{attribute 'GeneratedUsingTerminal: EK1100-0000-0018'}
{attribute addProperty BoxType "EK1100-0000-0018"}
{attribute addProperty Id "Beckhoff_EL1xxxEK1122Beckhoff_EL1xxxEK1122_4D1603AD2A_0001_EL1002_0000_0000EL1002_02444DCB6A_0002_EL1002_0000_0016EL1002_02444DCB6A_0003_EL1002_0000_0017EL1002_02444DCB6A_0004_EL1002_0000_0018EL1002_02444DCB6A_0005_EL1004_0000_0000EL1004_D135F8DB8A_0006_EL1004_0000_0016EL1004_D135F8DB8A_0007_EL1004_0000_0017EL1004_D135F8DB8A_0008_EL1004_0000_0018EL1004_D135F8DB8A_0009_EL1004_0000_0019EL1004_D135F8DB8A_0010_EL1004_0010_0000EL1004_D135F8DB8A_0011_EL1004_0010_0016EL1004_D135F8DB8A_0012_EL1004_0010_0017EL1004_D135F8DB8A_0013_EL1004_0010_0018EL1004_D135F8DB8A_0014_EL1004_0020_0016EL1004_D135F8DB8A_0015_EL1008_0000_0016EL1008_78E8D3DD12A_0016_EL1008_0000_0017EL1008_78E8D3DD12A_0017_EL1008_0000_0018EL1008_78E8D3DD12A_0018_EL1012_0000_0000EL1012_02444DCB6A_0019_EL1012_0000_0016EL1012_02444DCB6A_0020_EL1012_0000_0017EL1012_02444DCB6A_0021_EL1012_0000_0018EL1012_02444DCB6A_0022_EL1014_0000_0000EL1014_D135F8DB8A_0023_EL1014_0000_0016EL1014_D135F8DB8A_0024_EL1014_0000_0017EL1014_D135F8DB8A_0025_EL1014_0000_0018EL1014_D135F8DB8A_0026_EL1014_0000_0019EL1014_D135F8DB8A_0027_EL1014_0010_0000EL1014_D135F8DB8A_0028_EL1014_0010_0016EL1014_D135F8DB8A_0029_EL1014_0010_0017EL1014_D135F8DB8A_0030_EL1014_0010_0018EL1014_D135F8DB8A_0031_EL1014_0010_0019EL1014_D135F8DB8A_0032_EL1018_0000_0016EL1018_78E8D3DD12A_0033_EL1018_0000_0017EL1018_78E8D3DD12A_0034_EL1018_0000_0018EL1018_78E8D3DD12A_0035_EL1024_0000_0016EL1024_D135F8DB8A_0036_EL1024_0000_0017EL1024_D135F8DB8A_0037_EL1024_0000_0018EL1024_D135F8DB8A_0038_EL1034_0000_0016EL1034_D135F8DB8A_0039_EL1034_0000_0017EL1034_D135F8DB8A_0040_EL1034_0000_0018EL1034_D135F8DB8A_0041_EL1052_0000_0016EL1052_6CC2DB6A8A_0042_EL1054_0000_0016EL1054_37C87A1C12A_0043_EL1084_0000_0016EL1084_D135F8DB8A_0044_EL1084_0000_0017EL1084_D135F8DB8A_0045_EL1084_0000_0018EL1084_D135F8DB8A_0046_EL1088_0000_0016EL1088_78E8D3DD12A_0047_EL1088_0000_0017EL1088_78E8D3DD12A_0048_EL1088_0000_0018EL1088_78E8D3DD12A_0049_EL1094_0000_0016EL1094_D135F8DB8A_0050_EL1094_0000_0017EL1094_D135F8DB8A_0051_EL1094_0000_0018EL1094_D135F8DB8A_0052_EL1098_0000_0016EL1098_78E8D3DD12A_0053_EL1098_0000_0017EL1098_78E8D3DD12A_0054_EL1098_0000_0018EL1098_78E8D3DD12A_0055_EL1104_0000_0016EL1104_D135F8DB8A_0056_EL1104_0000_0017EL1104_D135F8DB8A_0057_EL1104_0000_0018EL1104_D135F8DB8A_0058_EL1114_0000_0016EL1114_D135F8DB8A_0059_EL1114_0000_0017EL1114_D135F8DB8A_0060_EL1114_0000_0018EL1114_D135F8DB8A_0061_EL1124_0000_0016EL1124_D135F8DB8A_0062_EL1124_0000_0017EL1124_D135F8DB8A_0063_EL1124_0000_0018EL1124_D135F8DB8A_0064_EL1134_0000_0016EL1134_D135F8DB8A_0065_EL1134_0000_0017EL1134_D135F8DB8A_0066_EL1134_0000_0018EL1134_D135F8DB8A_0067_EL1144_0000_0016EL1144_D135F8DB8A_0068_EL1144_0000_0017EL1144_D135F8DB8A_0069_EL1144_0000_0018EL1144_D135F8DB8A_0070_EL1202_0000_0016EL1202_02444DCB6A_0071_EL1202_0000_0017EL1202_02444DCB6A_0072_EL1202_0000_0018EL1202_02444DCB6A_0073_EL1202_0000_0019EL1202_02444DCB6A_0074_EL1202_0100_0016EL1202_647E460722A_0075_EL1202_0100_0017EL1202_647E460722A_0076_EL1202_0100_0018EL1202_647E460722A_0077_EL1202_0100_0019EL1202_647E460722A_0078_EL1252_0000_0017EL1252_0C2D47B448A_0079_EL1252_0000_0018EL1252_934A18FC48A_0080_EL1252_0000_0019EL1252_934A18FC48A_0081_EL1252_0000_0020EL1252_934A18FC48A_0082_EL1252_0000_0021EL1252_934A18FC48A_0083_EL1252_0000_0022EL1252_934A18FC48A_0084_EL1252_0010_0019EL1252_934A18FC48A_0085_EL1252_0010_0020EL1252_934A18FC48A_0086_EL1252_0010_0021EL1252_934A18FC48A_0087_EL1252_0050_0016EL1252_934A18FC48A_0088_EL1252_0050_0017EL1252_934A18FC48A_0089_EL1252_0050_0018EL1252_934A18FC48A_0090_EL1254_0000_0000EL1254_D5E6FA5F84A_0091_EL1262_0000_0002EL1262_0FA571DE40A_0092_EL1262_0000_0003EL1262_0FA571DE40A_0093_EL1262_0050_0002EL1262_0FA571DE40A_0094_EL1262_0050_0003EL1262_0FA571DE40A_0095_EL1258_0000_0016EL1258_FA676B82476A_0096_EL1258_0000_0017EL1258_FA676B82476A_0097_EL1258_0010_0017EL1258_E0C61872116A_0098_EL1259_0000_0016EL1259_D83D5EFD964A_0099_EL1259_0000_0017EL1259_22458C8C972A_0100_EL1259_0000_0018EL1259_22458C8C972A_0101_EL1382_0000_0016EL1382_6CC2DB6A8A_0102_EL1382_0000_0017EL1382_6CC2DB6A8A_0103_EL1382_0000_0018EL1382_6CC2DB6A8A_0104_EL1702_0000_0016EL1702_02444DCB6A_0105_EL1702_0000_0017EL1702_02444DCB6A_0106_EL1702_0020_0016EL1702_02444DCB6A_0107_EL1712_0000_0016EL1712_02444DCB6A_0108_EL1712_0020_0016EL1712_02444DCB6A_0109_EL1722_0000_0016EL1722_02444DCB6A_0110_EL1722_0000_0017EL1722_02444DCB6A_0111_EL1804_0000_0016EL1804_D135F8DB8A_0112_EL1804_0000_0017EL1804_D135F8DB8A_0113_EL1804_0000_0018EL1804_D135F8DB8A_0114_EL1808_0000_0016EL1808_78E8D3DD12A_0115_EL1808_0000_0017EL1808_78E8D3DD12A_0116_EL1808_0000_0018EL1808_78E8D3DD12A_0117_EL1809_0000_0016EL1809_32157CFD20A_0118_EL1809_0000_0017EL1809_32157CFD20A_0119_EL1809_0000_0018EL1809_32157CFD20A_0120_EL1814_0000_0016EL1814_D135F8DB8A_0121_EL1814_0000_0017EL1814_D135F8DB8A_0122_EL1814_0000_0018EL1814_D135F8DB8A_0123_EL1819_0000_0016EL1819_32157CFD20A_0124_EL1819_0000_0017EL1819_32157CFD20A_0125_EL1819_0000_0018EL1819_32157CFD20A_0126_EL1852_0000_0016EL1852_7699BCF620A_0127_EL1859_0000_0016EL1859_7699BCF620A_0128_EL1859_0000_0017EL1859_7699BCF620A_0129_EL1859_0000_0018EL1859_7699BCF620A_0130_EL1862_0000_0016EL1862_32157CFD20A_0131_EL1862_0000_0017EL1862_32157CFD20A_0132_EL1862_0000_0018EL1862_32157CFD20A_0133_EL1862_0000_0019EL1862_32157CFD20A_0134_EL1862_0010_0016EL1862_32157CFD20A_0135_EL1862_0010_0017EL1862_32157CFD20A_0136_EL1862_0010_0018EL1862_32157CFD20A_0137_EL1862_0010_0019EL1862_32157CFD20A_0138_EL1872_0000_0016EL1872_32157CFD20A_0139_EL1872_0000_0017EL1872_32157CFD20A_0140_EL1872_0000_0018EL1872_32157CFD20A_0141_EL1872_0010_0016EL1872_32157CFD20A_0142_EL1889_0000_0016EL1889_32157CFD20A_0143_EL1889_0000_0017EL1889_32157CFD20A_0144_EL1889_0000_0018EL1889_32157CFD20A_0145_EL1889_0000_0019EL1889_32157CFD20A_0146_EL1899_0000_0016EL1899_32157CFD20"}
{attribute addProperty CRC "3845396967"}
{attribute addProperty Size "6188"}
TYPE Beckhoff_EL1xxx_E53419E7 EXTENDS EK1100_1FC0878B :
STRUCT
	{attribute addProperty Name "Beckhoff_EL1xxxEK1122"}
	{attribute addProperty PreviousPort "Beckhoff EL1xxx : B"}
	Beckhoff_EL1xxxEK1122 : Beckhoff_EL1xxxEK1122_4D1603AD;
	{attribute addProperty Name "A_0001_EL1002_0000_0000"}
	{attribute addProperty PreviousPort "Beckhoff EL1xxxEK1122 : C"}
	A_0001_EL1002_0000_0000 : EL1002_02444DCB;
	{attribute addProperty Name "A_0002_EL1002_0000_0016"}
	{attribute addProperty PreviousPort "A_0001(EL1002-0000-0000) : B"}
	A_0002_EL1002_0000_0016 : EL1002_02444DCB;
	{attribute addProperty Name "A_0003_EL1002_0000_0017"}
	{attribute addProperty PreviousPort "A_0002(EL1002-0000-0016) : B"}
	A_0003_EL1002_0000_0017 : EL1002_02444DCB;
	{attribute addProperty Name "A_0004_EL1002_0000_0018"}
	{attribute addProperty PreviousPort "A_0003(EL1002-0000-0017) : B"}
	A_0004_EL1002_0000_0018 : EL1002_02444DCB;
	{attribute addProperty Name "A_0005_EL1004_0000_0000"}
	{attribute addProperty PreviousPort "A_0004(EL1002-0000-0018) : B"}
	A_0005_EL1004_0000_0000 : EL1004_D135F8DB;
	{attribute addProperty Name "A_0006_EL1004_0000_0016"}
	{attribute addProperty PreviousPort "A_0005(EL1004-0000-0000) : B"}
	A_0006_EL1004_0000_0016 : EL1004_D135F8DB;
	{attribute addProperty Name "A_0007_EL1004_0000_0017"}
	{attribute addProperty PreviousPort "A_0006(EL1004-0000-0016) : B"}
	A_0007_EL1004_0000_0017 : EL1004_D135F8DB;
	{attribute addProperty Name "A_0008_EL1004_0000_0018"}
	{attribute addProperty PreviousPort "A_0007(EL1004-0000-0017) : B"}
	A_0008_EL1004_0000_0018 : EL1004_D135F8DB;
	{attribute addProperty Name "A_0009_EL1004_0000_0019"}
	{attribute addProperty PreviousPort "A_0008(EL1004-0000-0018) : B"}
	A_0009_EL1004_0000_0019 : EL1004_D135F8DB;
	{attribute addProperty Name "A_0010_EL1004_0010_0000"}
	{attribute addProperty PreviousPort "A_0009(EL1004-0000-0019) : B"}
	A_0010_EL1004_0010_0000 : EL1004_D135F8DB;
	{attribute addProperty Name "A_0011_EL1004_0010_0016"}
	{attribute addProperty PreviousPort "A_0010(EL1004-0010-0000) : B"}
	A_0011_EL1004_0010_0016 : EL1004_D135F8DB;
	{attribute addProperty Name "A_0012_EL1004_0010_0017"}
	{attribute addProperty PreviousPort "A_0011(EL1004-0010-0016) : B"}
	A_0012_EL1004_0010_0017 : EL1004_D135F8DB;
	{attribute addProperty Name "A_0013_EL1004_0010_0018"}
	{attribute addProperty PreviousPort "A_0012(EL1004-0010-0017) : B"}
	A_0013_EL1004_0010_0018 : EL1004_D135F8DB;
	{attribute addProperty Name "A_0014_EL1004_0020_0016"}
	{attribute addProperty PreviousPort "A_0013(EL1004-0010-0018) : B"}
	A_0014_EL1004_0020_0016 : EL1004_D135F8DB;
	{attribute addProperty Name "A_0015_EL1008_0000_0016"}
	{attribute addProperty PreviousPort "A_0014(EL1004-0020-0016) : B"}
	A_0015_EL1008_0000_0016 : EL1008_78E8D3DD;
	{attribute addProperty Name "A_0016_EL1008_0000_0017"}
	{attribute addProperty PreviousPort "A_0015(EL1008-0000-0016) : B"}
	A_0016_EL1008_0000_0017 : EL1008_78E8D3DD;
	{attribute addProperty Name "A_0017_EL1008_0000_0018"}
	{attribute addProperty PreviousPort "A_0016(EL1008-0000-0017) : B"}
	A_0017_EL1008_0000_0018 : EL1008_78E8D3DD;
	{attribute addProperty Name "A_0018_EL1012_0000_0000"}
	{attribute addProperty PreviousPort "A_0017(EL1008-0000-0018) : B"}
	A_0018_EL1012_0000_0000 : EL1012_02444DCB;
	{attribute addProperty Name "A_0019_EL1012_0000_0016"}
	{attribute addProperty PreviousPort "A_0018(EL1012-0000-0000) : B"}
	A_0019_EL1012_0000_0016 : EL1012_02444DCB;
	{attribute addProperty Name "A_0020_EL1012_0000_0017"}
	{attribute addProperty PreviousPort "A_0019(EL1012-0000-0016) : B"}
	A_0020_EL1012_0000_0017 : EL1012_02444DCB;
	{attribute addProperty Name "A_0021_EL1012_0000_0018"}
	{attribute addProperty PreviousPort "A_0020(EL1012-0000-0017) : B"}
	A_0021_EL1012_0000_0018 : EL1012_02444DCB;
	{attribute addProperty Name "A_0022_EL1014_0000_0000"}
	{attribute addProperty PreviousPort "A_0021(EL1012-0000-0018) : B"}
	A_0022_EL1014_0000_0000 : EL1014_D135F8DB;
	{attribute addProperty Name "A_0023_EL1014_0000_0016"}
	{attribute addProperty PreviousPort "A_0022(EL1014-0000-0000) : B"}
	A_0023_EL1014_0000_0016 : EL1014_D135F8DB;
	{attribute addProperty Name "A_0024_EL1014_0000_0017"}
	{attribute addProperty PreviousPort "A_0023(EL1014-0000-0016) : B"}
	A_0024_EL1014_0000_0017 : EL1014_D135F8DB;
	{attribute addProperty Name "A_0025_EL1014_0000_0018"}
	{attribute addProperty PreviousPort "A_0024(EL1014-0000-0017) : B"}
	A_0025_EL1014_0000_0018 : EL1014_D135F8DB;
	{attribute addProperty Name "A_0026_EL1014_0000_0019"}
	{attribute addProperty PreviousPort "A_0025(EL1014-0000-0018) : B"}
	A_0026_EL1014_0000_0019 : EL1014_D135F8DB;
	{attribute addProperty Name "A_0027_EL1014_0010_0000"}
	{attribute addProperty PreviousPort "A_0026(EL1014-0000-0019) : B"}
	A_0027_EL1014_0010_0000 : EL1014_D135F8DB;
	{attribute addProperty Name "A_0028_EL1014_0010_0016"}
	{attribute addProperty PreviousPort "A_0027(EL1014-0010-0000) : B"}
	A_0028_EL1014_0010_0016 : EL1014_D135F8DB;
	{attribute addProperty Name "A_0029_EL1014_0010_0017"}
	{attribute addProperty PreviousPort "A_0028(EL1014-0010-0016) : B"}
	A_0029_EL1014_0010_0017 : EL1014_D135F8DB;
	{attribute addProperty Name "A_0030_EL1014_0010_0018"}
	{attribute addProperty PreviousPort "A_0029(EL1014-0010-0017) : B"}
	A_0030_EL1014_0010_0018 : EL1014_D135F8DB;
	{attribute addProperty Name "A_0031_EL1014_0010_0019"}
	{attribute addProperty PreviousPort "A_0030(EL1014-0010-0018) : B"}
	A_0031_EL1014_0010_0019 : EL1014_D135F8DB;
	{attribute addProperty Name "A_0032_EL1018_0000_0016"}
	{attribute addProperty PreviousPort "A_0031(EL1014-0010-0019) : B"}
	A_0032_EL1018_0000_0016 : EL1018_78E8D3DD;
	{attribute addProperty Name "A_0033_EL1018_0000_0017"}
	{attribute addProperty PreviousPort "A_0032(EL1018-0000-0016) : B"}
	A_0033_EL1018_0000_0017 : EL1018_78E8D3DD;
	{attribute addProperty Name "A_0034_EL1018_0000_0018"}
	{attribute addProperty PreviousPort "A_0033(EL1018-0000-0017) : B"}
	A_0034_EL1018_0000_0018 : EL1018_78E8D3DD;
	{attribute addProperty Name "A_0035_EL1024_0000_0016"}
	{attribute addProperty PreviousPort "A_0034(EL1018-0000-0018) : B"}
	A_0035_EL1024_0000_0016 : EL1024_D135F8DB;
	{attribute addProperty Name "A_0036_EL1024_0000_0017"}
	{attribute addProperty PreviousPort "A_0035(EL1024-0000-0016) : B"}
	A_0036_EL1024_0000_0017 : EL1024_D135F8DB;
	{attribute addProperty Name "A_0037_EL1024_0000_0018"}
	{attribute addProperty PreviousPort "A_0036(EL1024-0000-0017) : B"}
	A_0037_EL1024_0000_0018 : EL1024_D135F8DB;
	{attribute addProperty Name "A_0038_EL1034_0000_0016"}
	{attribute addProperty PreviousPort "A_0037(EL1024-0000-0018) : B"}
	A_0038_EL1034_0000_0016 : EL1034_D135F8DB;
	{attribute addProperty Name "A_0039_EL1034_0000_0017"}
	{attribute addProperty PreviousPort "A_0038(EL1034-0000-0016) : B"}
	A_0039_EL1034_0000_0017 : EL1034_D135F8DB;
	{attribute addProperty Name "A_0040_EL1034_0000_0018"}
	{attribute addProperty PreviousPort "A_0039(EL1034-0000-0017) : B"}
	A_0040_EL1034_0000_0018 : EL1034_D135F8DB;
	{attribute addProperty Name "A_0041_EL1052_0000_0016"}
	{attribute addProperty PreviousPort "A_0040(EL1034-0000-0018) : B"}
	A_0041_EL1052_0000_0016 : EL1052_6CC2DB6A;
	{attribute addProperty Name "A_0042_EL1054_0000_0016"}
	{attribute addProperty PreviousPort "A_0041(EL1052-0000-0016) : B"}
	A_0042_EL1054_0000_0016 : EL1054_37C87A1C;
	{attribute addProperty Name "A_0043_EL1084_0000_0016"}
	{attribute addProperty PreviousPort "A_0042(EL1054-0000-0016) : B"}
	A_0043_EL1084_0000_0016 : EL1084_D135F8DB;
	{attribute addProperty Name "A_0044_EL1084_0000_0017"}
	{attribute addProperty PreviousPort "A_0043(EL1084-0000-0016) : B"}
	A_0044_EL1084_0000_0017 : EL1084_D135F8DB;
	{attribute addProperty Name "A_0045_EL1084_0000_0018"}
	{attribute addProperty PreviousPort "A_0044(EL1084-0000-0017) : B"}
	A_0045_EL1084_0000_0018 : EL1084_D135F8DB;
	{attribute addProperty Name "A_0046_EL1088_0000_0016"}
	{attribute addProperty PreviousPort "A_0045(EL1084-0000-0018) : B"}
	A_0046_EL1088_0000_0016 : EL1088_78E8D3DD;
	{attribute addProperty Name "A_0047_EL1088_0000_0017"}
	{attribute addProperty PreviousPort "A_0046(EL1088-0000-0016) : B"}
	A_0047_EL1088_0000_0017 : EL1088_78E8D3DD;
	{attribute addProperty Name "A_0048_EL1088_0000_0018"}
	{attribute addProperty PreviousPort "A_0047(EL1088-0000-0017) : B"}
	A_0048_EL1088_0000_0018 : EL1088_78E8D3DD;
	{attribute addProperty Name "A_0049_EL1094_0000_0016"}
	{attribute addProperty PreviousPort "A_0048(EL1088-0000-0018) : B"}
	A_0049_EL1094_0000_0016 : EL1094_D135F8DB;
	{attribute addProperty Name "A_0050_EL1094_0000_0017"}
	{attribute addProperty PreviousPort "A_0049(EL1094-0000-0016) : B"}
	A_0050_EL1094_0000_0017 : EL1094_D135F8DB;
	{attribute addProperty Name "A_0051_EL1094_0000_0018"}
	{attribute addProperty PreviousPort "A_0050(EL1094-0000-0017) : B"}
	A_0051_EL1094_0000_0018 : EL1094_D135F8DB;
	{attribute addProperty Name "A_0052_EL1098_0000_0016"}
	{attribute addProperty PreviousPort "A_0051(EL1094-0000-0018) : B"}
	A_0052_EL1098_0000_0016 : EL1098_78E8D3DD;
	{attribute addProperty Name "A_0053_EL1098_0000_0017"}
	{attribute addProperty PreviousPort "A_0052(EL1098-0000-0016) : B"}
	A_0053_EL1098_0000_0017 : EL1098_78E8D3DD;
	{attribute addProperty Name "A_0054_EL1098_0000_0018"}
	{attribute addProperty PreviousPort "A_0053(EL1098-0000-0017) : B"}
	A_0054_EL1098_0000_0018 : EL1098_78E8D3DD;
	{attribute addProperty Name "A_0055_EL1104_0000_0016"}
	{attribute addProperty PreviousPort "A_0054(EL1098-0000-0018) : B"}
	A_0055_EL1104_0000_0016 : EL1104_D135F8DB;
	{attribute addProperty Name "A_0056_EL1104_0000_0017"}
	{attribute addProperty PreviousPort "A_0055(EL1104-0000-0016) : B"}
	A_0056_EL1104_0000_0017 : EL1104_D135F8DB;
	{attribute addProperty Name "A_0057_EL1104_0000_0018"}
	{attribute addProperty PreviousPort "A_0056(EL1104-0000-0017) : B"}
	A_0057_EL1104_0000_0018 : EL1104_D135F8DB;
	{attribute addProperty Name "A_0058_EL1114_0000_0016"}
	{attribute addProperty PreviousPort "A_0057(EL1104-0000-0018) : B"}
	A_0058_EL1114_0000_0016 : EL1114_D135F8DB;
	{attribute addProperty Name "A_0059_EL1114_0000_0017"}
	{attribute addProperty PreviousPort "A_0058(EL1114-0000-0016) : B"}
	A_0059_EL1114_0000_0017 : EL1114_D135F8DB;
	{attribute addProperty Name "A_0060_EL1114_0000_0018"}
	{attribute addProperty PreviousPort "A_0059(EL1114-0000-0017) : B"}
	A_0060_EL1114_0000_0018 : EL1114_D135F8DB;
	{attribute addProperty Name "A_0061_EL1124_0000_0016"}
	{attribute addProperty PreviousPort "A_0060(EL1114-0000-0018) : B"}
	A_0061_EL1124_0000_0016 : EL1124_D135F8DB;
	{attribute addProperty Name "A_0062_EL1124_0000_0017"}
	{attribute addProperty PreviousPort "A_0061(EL1124-0000-0016) : B"}
	A_0062_EL1124_0000_0017 : EL1124_D135F8DB;
	{attribute addProperty Name "A_0063_EL1124_0000_0018"}
	{attribute addProperty PreviousPort "A_0062(EL1124-0000-0017) : B"}
	A_0063_EL1124_0000_0018 : EL1124_D135F8DB;
	{attribute addProperty Name "A_0064_EL1134_0000_0016"}
	{attribute addProperty PreviousPort "A_0063(EL1124-0000-0018) : B"}
	A_0064_EL1134_0000_0016 : EL1134_D135F8DB;
	{attribute addProperty Name "A_0065_EL1134_0000_0017"}
	{attribute addProperty PreviousPort "A_0064(EL1134-0000-0016) : B"}
	A_0065_EL1134_0000_0017 : EL1134_D135F8DB;
	{attribute addProperty Name "A_0066_EL1134_0000_0018"}
	{attribute addProperty PreviousPort "A_0065(EL1134-0000-0017) : B"}
	A_0066_EL1134_0000_0018 : EL1134_D135F8DB;
	{attribute addProperty Name "A_0067_EL1144_0000_0016"}
	{attribute addProperty PreviousPort "A_0066(EL1134-0000-0018) : B"}
	A_0067_EL1144_0000_0016 : EL1144_D135F8DB;
	{attribute addProperty Name "A_0068_EL1144_0000_0017"}
	{attribute addProperty PreviousPort "A_0067(EL1144-0000-0016) : B"}
	A_0068_EL1144_0000_0017 : EL1144_D135F8DB;
	{attribute addProperty Name "A_0069_EL1144_0000_0018"}
	{attribute addProperty PreviousPort "A_0068(EL1144-0000-0017) : B"}
	A_0069_EL1144_0000_0018 : EL1144_D135F8DB;
	{attribute addProperty Name "A_0070_EL1202_0000_0016"}
	{attribute addProperty PreviousPort "A_0069(EL1144-0000-0018) : B"}
	A_0070_EL1202_0000_0016 : EL1202_02444DCB;
	{attribute addProperty Name "A_0071_EL1202_0000_0017"}
	{attribute addProperty PreviousPort "A_0070(EL1202-0000-0016) : B"}
	A_0071_EL1202_0000_0017 : EL1202_02444DCB;
	{attribute addProperty Name "A_0072_EL1202_0000_0018"}
	{attribute addProperty PreviousPort "A_0071(EL1202-0000-0017) : B"}
	A_0072_EL1202_0000_0018 : EL1202_02444DCB;
	{attribute addProperty Name "A_0073_EL1202_0000_0019"}
	{attribute addProperty PreviousPort "A_0072(EL1202-0000-0018) : B"}
	A_0073_EL1202_0000_0019 : EL1202_02444DCB;
	{attribute addProperty Name "A_0074_EL1202_0100_0016"}
	{attribute addProperty PreviousPort "A_0073(EL1202-0000-0019) : B"}
	A_0074_EL1202_0100_0016 : EL1202_647E4607;
	{attribute addProperty Name "A_0075_EL1202_0100_0017"}
	{attribute addProperty PreviousPort "A_0074(EL1202-0100-0016) : B"}
	A_0075_EL1202_0100_0017 : EL1202_647E4607;
	{attribute addProperty Name "A_0076_EL1202_0100_0018"}
	{attribute addProperty PreviousPort "A_0075(EL1202-0100-0017) : B"}
	A_0076_EL1202_0100_0018 : EL1202_647E4607;
	{attribute addProperty Name "A_0077_EL1202_0100_0019"}
	{attribute addProperty PreviousPort "A_0076(EL1202-0100-0018) : B"}
	A_0077_EL1202_0100_0019 : EL1202_647E4607;
	{attribute addProperty Name "A_0078_EL1252_0000_0017"}
	{attribute addProperty PreviousPort "A_0077(EL1202-0100-0019) : B"}
	A_0078_EL1252_0000_0017 : EL1252_0C2D47B4;
	{attribute addProperty Name "A_0079_EL1252_0000_0018"}
	{attribute addProperty PreviousPort "A_0078(EL1252-0000-0017) : B"}
	A_0079_EL1252_0000_0018 : EL1252_934A18FC;
	{attribute addProperty Name "A_0080_EL1252_0000_0019"}
	{attribute addProperty PreviousPort "A_0079(EL1252-0000-0018) : B"}
	A_0080_EL1252_0000_0019 : EL1252_934A18FC;
	{attribute addProperty Name "A_0081_EL1252_0000_0020"}
	{attribute addProperty PreviousPort "A_0080(EL1252-0000-0019) : B"}
	A_0081_EL1252_0000_0020 : EL1252_934A18FC;
	{attribute addProperty Name "A_0082_EL1252_0000_0021"}
	{attribute addProperty PreviousPort "A_0081(EL1252-0000-0020) : B"}
	A_0082_EL1252_0000_0021 : EL1252_934A18FC;
	{attribute addProperty Name "A_0083_EL1252_0000_0022"}
	{attribute addProperty PreviousPort "A_0082(EL1252-0000-0021) : B"}
	A_0083_EL1252_0000_0022 : EL1252_934A18FC;
	{attribute addProperty Name "A_0084_EL1252_0010_0019"}
	{attribute addProperty PreviousPort "A_0083(EL1252-0000-0022) : B"}
	A_0084_EL1252_0010_0019 : EL1252_934A18FC;
	{attribute addProperty Name "A_0085_EL1252_0010_0020"}
	{attribute addProperty PreviousPort "A_0084(EL1252-0010-0019) : B"}
	A_0085_EL1252_0010_0020 : EL1252_934A18FC;
	{attribute addProperty Name "A_0086_EL1252_0010_0021"}
	{attribute addProperty PreviousPort "A_0085(EL1252-0010-0020) : B"}
	A_0086_EL1252_0010_0021 : EL1252_934A18FC;
	{attribute addProperty Name "A_0087_EL1252_0050_0016"}
	{attribute addProperty PreviousPort "A_0086(EL1252-0010-0021) : B"}
	A_0087_EL1252_0050_0016 : EL1252_934A18FC;
	{attribute addProperty Name "A_0088_EL1252_0050_0017"}
	{attribute addProperty PreviousPort "A_0087(EL1252-0050-0016) : B"}
	A_0088_EL1252_0050_0017 : EL1252_934A18FC;
	{attribute addProperty Name "A_0089_EL1252_0050_0018"}
	{attribute addProperty PreviousPort "A_0088(EL1252-0050-0017) : B"}
	A_0089_EL1252_0050_0018 : EL1252_934A18FC;
	{attribute addProperty Name "A_0090_EL1254_0000_0000"}
	{attribute addProperty PreviousPort "A_0089(EL1252-0050-0018) : B"}
	A_0090_EL1254_0000_0000 : EL1254_D5E6FA5F;
	{attribute addProperty Name "A_0091_EL1262_0000_0002"}
	{attribute addProperty PreviousPort "A_0090(EL1254-0000-0000) : B"}
	A_0091_EL1262_0000_0002 : EL1262_0FA571DE;
	{attribute addProperty Name "A_0092_EL1262_0000_0003"}
	{attribute addProperty PreviousPort "A_0091(EL1262-0000-0002) : B"}
	A_0092_EL1262_0000_0003 : EL1262_0FA571DE;
	{attribute addProperty Name "A_0093_EL1262_0050_0002"}
	{attribute addProperty PreviousPort "A_0092(EL1262-0000-0003) : B"}
	A_0093_EL1262_0050_0002 : EL1262_0FA571DE;
	{attribute addProperty Name "A_0094_EL1262_0050_0003"}
	{attribute addProperty PreviousPort "A_0093(EL1262-0050-0002) : B"}
	A_0094_EL1262_0050_0003 : EL1262_0FA571DE;
	{attribute addProperty Name "A_0095_EL1258_0000_0016"}
	{attribute addProperty PreviousPort "A_0094(EL1262-0050-0003) : B"}
	A_0095_EL1258_0000_0016 : EL1258_FA676B82;
	{attribute addProperty Name "A_0096_EL1258_0000_0017"}
	{attribute addProperty PreviousPort "A_0095(EL1258-0000-0016) : B"}
	A_0096_EL1258_0000_0017 : EL1258_FA676B82;
	{attribute addProperty Name "A_0097_EL1258_0010_0017"}
	{attribute addProperty PreviousPort "A_0096(EL1258-0000-0017) : B"}
	A_0097_EL1258_0010_0017 : EL1258_E0C61872;
	{attribute addProperty Name "A_0098_EL1259_0000_0016"}
	{attribute addProperty PreviousPort "A_0097(EL1258-0010-0017) : B"}
	A_0098_EL1259_0000_0016 : EL1259_D83D5EFD;
	{attribute addProperty Name "A_0099_EL1259_0000_0017"}
	{attribute addProperty PreviousPort "A_0098(EL1259-0000-0016) : B"}
	A_0099_EL1259_0000_0017 : EL1259_22458C8C;
	{attribute addProperty Name "A_0100_EL1259_0000_0018"}
	{attribute addProperty PreviousPort "A_0099(EL1259-0000-0017) : B"}
	A_0100_EL1259_0000_0018 : EL1259_22458C8C;
	{attribute addProperty Name "A_0101_EL1382_0000_0016"}
	{attribute addProperty PreviousPort "A_0100(EL1259-0000-0018) : B"}
	A_0101_EL1382_0000_0016 : EL1382_6CC2DB6A;
	{attribute addProperty Name "A_0102_EL1382_0000_0017"}
	{attribute addProperty PreviousPort "A_0101(EL1382-0000-0016) : B"}
	A_0102_EL1382_0000_0017 : EL1382_6CC2DB6A;
	{attribute addProperty Name "A_0103_EL1382_0000_0018"}
	{attribute addProperty PreviousPort "A_0102(EL1382-0000-0017) : B"}
	A_0103_EL1382_0000_0018 : EL1382_6CC2DB6A;
	{attribute addProperty Name "A_0104_EL1702_0000_0016"}
	{attribute addProperty PreviousPort "A_0103(EL1382-0000-0018) : B"}
	A_0104_EL1702_0000_0016 : EL1702_02444DCB;
	{attribute addProperty Name "A_0105_EL1702_0000_0017"}
	{attribute addProperty PreviousPort "A_0104(EL1702-0000-0016) : B"}
	A_0105_EL1702_0000_0017 : EL1702_02444DCB;
	{attribute addProperty Name "A_0106_EL1702_0020_0016"}
	{attribute addProperty PreviousPort "A_0105(EL1702-0000-0017) : B"}
	A_0106_EL1702_0020_0016 : EL1702_02444DCB;
	{attribute addProperty Name "A_0107_EL1712_0000_0016"}
	{attribute addProperty PreviousPort "A_0106(EL1702-0020-0016) : B"}
	A_0107_EL1712_0000_0016 : EL1712_02444DCB;
	{attribute addProperty Name "A_0108_EL1712_0020_0016"}
	{attribute addProperty PreviousPort "A_0107(EL1712-0000-0016) : B"}
	A_0108_EL1712_0020_0016 : EL1712_02444DCB;
	{attribute addProperty Name "A_0109_EL1722_0000_0016"}
	{attribute addProperty PreviousPort "A_0108(EL1712-0020-0016) : B"}
	A_0109_EL1722_0000_0016 : EL1722_02444DCB;
	{attribute addProperty Name "A_0110_EL1722_0000_0017"}
	{attribute addProperty PreviousPort "A_0109(EL1722-0000-0016) : B"}
	A_0110_EL1722_0000_0017 : EL1722_02444DCB;
	{attribute addProperty Name "A_0111_EL1804_0000_0016"}
	{attribute addProperty PreviousPort "A_0110(EL1722-0000-0017) : B"}
	A_0111_EL1804_0000_0016 : EL1804_D135F8DB;
	{attribute addProperty Name "A_0112_EL1804_0000_0017"}
	{attribute addProperty PreviousPort "A_0111(EL1804-0000-0016) : B"}
	A_0112_EL1804_0000_0017 : EL1804_D135F8DB;
	{attribute addProperty Name "A_0113_EL1804_0000_0018"}
	{attribute addProperty PreviousPort "A_0112(EL1804-0000-0017) : B"}
	A_0113_EL1804_0000_0018 : EL1804_D135F8DB;
	{attribute addProperty Name "A_0114_EL1808_0000_0016"}
	{attribute addProperty PreviousPort "A_0113(EL1804-0000-0018) : B"}
	A_0114_EL1808_0000_0016 : EL1808_78E8D3DD;
	{attribute addProperty Name "A_0115_EL1808_0000_0017"}
	{attribute addProperty PreviousPort "A_0114(EL1808-0000-0016) : B"}
	A_0115_EL1808_0000_0017 : EL1808_78E8D3DD;
	{attribute addProperty Name "A_0116_EL1808_0000_0018"}
	{attribute addProperty PreviousPort "A_0115(EL1808-0000-0017) : B"}
	A_0116_EL1808_0000_0018 : EL1808_78E8D3DD;
	{attribute addProperty Name "A_0117_EL1809_0000_0016"}
	{attribute addProperty PreviousPort "A_0116(EL1808-0000-0018) : B"}
	A_0117_EL1809_0000_0016 : EL1809_32157CFD;
	{attribute addProperty Name "A_0118_EL1809_0000_0017"}
	{attribute addProperty PreviousPort "A_0117(EL1809-0000-0016) : B"}
	A_0118_EL1809_0000_0017 : EL1809_32157CFD;
	{attribute addProperty Name "A_0119_EL1809_0000_0018"}
	{attribute addProperty PreviousPort "A_0118(EL1809-0000-0017) : B"}
	A_0119_EL1809_0000_0018 : EL1809_32157CFD;
	{attribute addProperty Name "A_0120_EL1814_0000_0016"}
	{attribute addProperty PreviousPort "A_0119(EL1809-0000-0018) : B"}
	A_0120_EL1814_0000_0016 : EL1814_D135F8DB;
	{attribute addProperty Name "A_0121_EL1814_0000_0017"}
	{attribute addProperty PreviousPort "A_0120(EL1814-0000-0016) : B"}
	A_0121_EL1814_0000_0017 : EL1814_D135F8DB;
	{attribute addProperty Name "A_0122_EL1814_0000_0018"}
	{attribute addProperty PreviousPort "A_0121(EL1814-0000-0017) : B"}
	A_0122_EL1814_0000_0018 : EL1814_D135F8DB;
	{attribute addProperty Name "A_0123_EL1819_0000_0016"}
	{attribute addProperty PreviousPort "A_0122(EL1814-0000-0018) : B"}
	A_0123_EL1819_0000_0016 : EL1819_32157CFD;
	{attribute addProperty Name "A_0124_EL1819_0000_0017"}
	{attribute addProperty PreviousPort "A_0123(EL1819-0000-0016) : B"}
	A_0124_EL1819_0000_0017 : EL1819_32157CFD;
	{attribute addProperty Name "A_0125_EL1819_0000_0018"}
	{attribute addProperty PreviousPort "A_0124(EL1819-0000-0017) : B"}
	A_0125_EL1819_0000_0018 : EL1819_32157CFD;
	{attribute addProperty Name "A_0126_EL1852_0000_0016"}
	{attribute addProperty PreviousPort "A_0125(EL1819-0000-0018) : B"}
	A_0126_EL1852_0000_0016 : EL1852_7699BCF6;
	{attribute addProperty Name "A_0127_EL1859_0000_0016"}
	{attribute addProperty PreviousPort "A_0126(EL1852-0000-0016) : B"}
	A_0127_EL1859_0000_0016 : EL1859_7699BCF6;
	{attribute addProperty Name "A_0128_EL1859_0000_0017"}
	{attribute addProperty PreviousPort "A_0127(EL1859-0000-0016) : B"}
	A_0128_EL1859_0000_0017 : EL1859_7699BCF6;
	{attribute addProperty Name "A_0129_EL1859_0000_0018"}
	{attribute addProperty PreviousPort "A_0128(EL1859-0000-0017) : B"}
	A_0129_EL1859_0000_0018 : EL1859_7699BCF6;
	{attribute addProperty Name "A_0130_EL1862_0000_0016"}
	{attribute addProperty PreviousPort "A_0129(EL1859-0000-0018) : B"}
	A_0130_EL1862_0000_0016 : EL1862_32157CFD;
	{attribute addProperty Name "A_0131_EL1862_0000_0017"}
	{attribute addProperty PreviousPort "A_0130(EL1862-0000-0016) : B"}
	A_0131_EL1862_0000_0017 : EL1862_32157CFD;
	{attribute addProperty Name "A_0132_EL1862_0000_0018"}
	{attribute addProperty PreviousPort "A_0131(EL1862-0000-0017) : B"}
	A_0132_EL1862_0000_0018 : EL1862_32157CFD;
	{attribute addProperty Name "A_0133_EL1862_0000_0019"}
	{attribute addProperty PreviousPort "A_0132(EL1862-0000-0018) : B"}
	A_0133_EL1862_0000_0019 : EL1862_32157CFD;
	{attribute addProperty Name "A_0134_EL1862_0010_0016"}
	{attribute addProperty PreviousPort "A_0133(EL1862-0000-0019) : B"}
	A_0134_EL1862_0010_0016 : EL1862_32157CFD;
	{attribute addProperty Name "A_0135_EL1862_0010_0017"}
	{attribute addProperty PreviousPort "A_0134(EL1862-0010-0016) : B"}
	A_0135_EL1862_0010_0017 : EL1862_32157CFD;
	{attribute addProperty Name "A_0136_EL1862_0010_0018"}
	{attribute addProperty PreviousPort "A_0135(EL1862-0010-0017) : B"}
	A_0136_EL1862_0010_0018 : EL1862_32157CFD;
	{attribute addProperty Name "A_0137_EL1862_0010_0019"}
	{attribute addProperty PreviousPort "A_0136(EL1862-0010-0018) : B"}
	A_0137_EL1862_0010_0019 : EL1862_32157CFD;
	{attribute addProperty Name "A_0138_EL1872_0000_0016"}
	{attribute addProperty PreviousPort "A_0137(EL1862-0010-0019) : B"}
	A_0138_EL1872_0000_0016 : EL1872_32157CFD;
	{attribute addProperty Name "A_0139_EL1872_0000_0017"}
	{attribute addProperty PreviousPort "A_0138(EL1872-0000-0016) : B"}
	A_0139_EL1872_0000_0017 : EL1872_32157CFD;
	{attribute addProperty Name "A_0140_EL1872_0000_0018"}
	{attribute addProperty PreviousPort "A_0139(EL1872-0000-0017) : B"}
	A_0140_EL1872_0000_0018 : EL1872_32157CFD;
	{attribute addProperty Name "A_0141_EL1872_0010_0016"}
	{attribute addProperty PreviousPort "A_0140(EL1872-0000-0018) : B"}
	A_0141_EL1872_0010_0016 : EL1872_32157CFD;
	{attribute addProperty Name "A_0142_EL1889_0000_0016"}
	{attribute addProperty PreviousPort "A_0141(EL1872-0010-0016) : B"}
	A_0142_EL1889_0000_0016 : EL1889_32157CFD;
	{attribute addProperty Name "A_0143_EL1889_0000_0017"}
	{attribute addProperty PreviousPort "A_0142(EL1889-0000-0016) : B"}
	A_0143_EL1889_0000_0017 : EL1889_32157CFD;
	{attribute addProperty Name "A_0144_EL1889_0000_0018"}
	{attribute addProperty PreviousPort "A_0143(EL1889-0000-0017) : B"}
	A_0144_EL1889_0000_0018 : EL1889_32157CFD;
	{attribute addProperty Name "A_0145_EL1889_0000_0019"}
	{attribute addProperty PreviousPort "A_0144(EL1889-0000-0018) : B"}
	A_0145_EL1889_0000_0019 : EL1889_32157CFD;
	{attribute addProperty Name "A_0146_EL1899_0000_0016"}
	{attribute addProperty PreviousPort "A_0145(EL1889-0000-0019) : B"}
	A_0146_EL1899_0000_0016 : EL1899_32157CFD;
END_STRUCT
END_TYPE

(* stored: Version 1.2.0.0, ProductVersion 3.1.4024.9
   DUT Beckhoff_EL1xxx_E53419E7: Id {99e1a61a-bb56-4e93-9486-a16e99ee82bb} *)
